TYPE ByteOr8Bits :
UNION
	Byte_ : BYTE;
	Bits8 : Bits8;
END_UNION
END_TYPE

(* stored: Version 1.1.0.1
   DUT ByteOr8Bits: Id {9e3ed942-6806-019f-1220-8db92fbb0955} *)
